DATA_BLOCK "MotorDB"
{ S7_Optimized_Access := 'TRUE'; DB_Accessible_From_OPC_UA := 'TRUE'; DB_Accessible_From_Webserver := 'TRUE' }
VERSION : '1.0'
VAR
    TEMPERATURE : REAL;
END_VAR

VAR RETAIN
    SPEED : INT;
    ACCELERATION : INT;
END_VAR
END_DATA_BLOCK